// ==============================================================================
// FC_HAL_Redler_Read - Читання HAL входів редлерів
// ==============================================================================
// Project  : Elevator_System
// Author   : Engineering Team
// Version  : 1.0.0
// Generated: 2026-01-14 10:18:12
// ==============================================================================

FUNCTION "FC_HAL_Redler_Read" : VOID
{ S7_Optimized_Access := 'TRUE' }
VERSION : 1.0

VAR_IN_OUT
    Redler : ARRAY[*] OF "UDT_Redler";
END_VAR

BEGIN
    // Редлер_1
    Redler[0].DI_Speed_OK    := "DB_HAL_Redler".DI_Speed_0;
    Redler[0].DI_Breaker_OK  := "DB_HAL_Redler".DI_Breaker_0;
    Redler[0].DI_Overflow_OK := "DB_HAL_Redler".DI_Overflow_0;

    // Редлер_2
    Redler[1].DI_Speed_OK    := "DB_HAL_Redler".DI_Speed_1;
    Redler[1].DI_Breaker_OK  := "DB_HAL_Redler".DI_Breaker_1;
    Redler[1].DI_Overflow_OK := "DB_HAL_Redler".DI_Overflow_1;

END_FUNCTION
